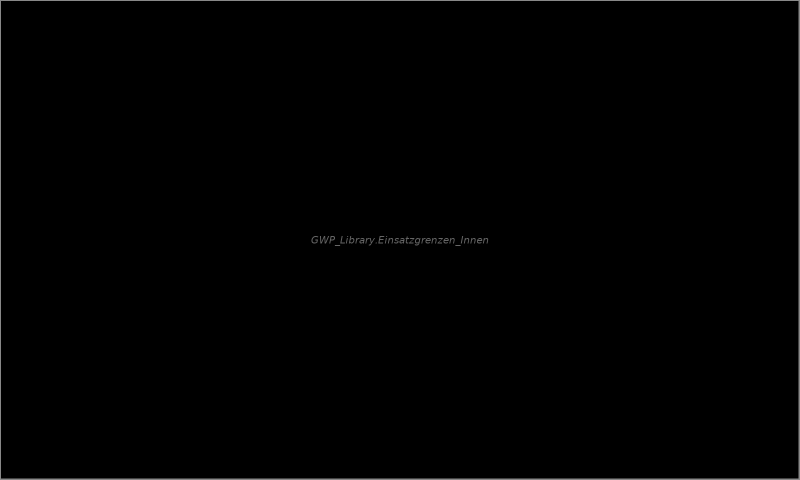
VISUALIZATION EG  // 800x480
    Frame (0,0 800x480)
        shows GWP_Library.Einsatzgrenzen_Innen(FB_Einsatzgrenzen_Innen := MAIN.Kreis_3KO_0.Einsatzgrenzen_Innen, FB_Init_1 := MAIN.Init_0)
END_VISUALIZATION

(* stored: Version 1.1.0.1, ProductVersion 3.1.4022.6
   Visu EG: Id {8c00dd7c-f5a6-4635-9cb0-308497526b56} *)
